// TwinCAT 3 PLC project Aufgabe_6
// ProgramVersion: 3.1.4022.3
// libraries:
//   Tc2_Standard, * (Beckhoff Automation GmbH)
//   Tc2_System, * (Beckhoff Automation GmbH)
//   Tc3_Module, * (Beckhoff Automation GmbH)
// project tree:
//   DUTs/ RS232_Return.TcDUT
//   / PlcTask.TcTTO
//   POUs/ MAIN.TcPOU, RS232.TcPOU
// (motion and I/O tree: see PLC project aufgabenserie2)
// real-time tasks:
//   TASK PlcTask: cycle T#10ms, priority 20, ADS port 350
// variable links:

CONFIGURATION Aufgabe_6
    RESOURCE PLC ON TwinCAT3
        TASK PlcTask(INTERVAL := T#10ms, PRIORITY := 20);
        PROGRAM MAIN WITH PlcTask : MAIN;
    END_RESOURCE
END_CONFIGURATION

// ---- DUTs/RS232_Return.TcDUT
TYPE RS232_Return :
STRUCT
	inLenght : INT;
	overrunError : BOOL;
	framingError : BOOL;
	parityError : BOOL;
	bufferFull : BOOL;
	initAccepted : BOOL;
	receiveRequest : BOOL;
	transmitAccepted : BOOL;
END_STRUCT
END_TYPE

// ---- POUs/MAIN.TcPOU
PROGRAM MAIN
VAR
	i_Result1 : RS232_Return;
	i_Result2 : RS232_Return;
	i_Result3 : RS232_Return;
END_VAR

i_Result1 := RS232(w_RS232Input:= 16#1D06);
i_Result2 := RS232(w_RS232Input:= 16#534C);
i_Result3 := RS232(w_RS232Input:= 16#C705);

END_PROGRAM

// ---- POUs/RS232.TcPOU
FUNCTION RS232 : RS232_Return
VAR_INPUT
	w_RS232Input : WORD;
END_VAR
VAR
	s_RS232Temp : RS232_Return;
END_VAR

s_RS232Temp.inLenght := WORD_TO_INT(SHR(w_RS232Input, 8));
s_RS232Temp.overrunError := WORD_TO_BOOL(SHL(1,6) AND w_RS232Input);
s_RS232Temp.framingError := WORD_TO_BOOL(SHL(1,5) AND w_RS232Input);
s_RS232Temp.parityError := WORD_TO_BOOL(SHL(1,4) AND w_RS232Input);
s_RS232Temp.bufferFull := WORD_TO_BOOL(SHL(1,3) AND w_RS232Input);
s_RS232Temp.initAccepted := WORD_TO_BOOL(SHL(1,2) AND w_RS232Input);
s_RS232Temp.receiveRequest := WORD_TO_BOOL(SHL(1,1) AND w_RS232Input);
s_RS232Temp.transmitAccepted := WORD_TO_BOOL(SHL(1,0) AND w_RS232Input);
RS232 := s_RS232Temp;

END_FUNCTION
